// TIA Portal V20 export
DATA_BLOCK "DB_Tracability"   // DB94
// stored: InstanceOfName FB_Tracability, InstanceOfType FB
"FB_Tracability"
   // VAR_INPUT
   //    iCondTransfertExtInTo1 : Bool;
   //    iCondTransfertExtInTo2 : Bool;
   //    iCondTransfert1To3 : Bool;
   //    iCondTransfert2To3 : Bool;
   //    iCondTransfert3To4 : Bool;
   //    iCondTransfert4To5 : Bool;
   //    iCondTransfert5To6 : Bool;
   //    iCondTransfert5To7 : Bool;
   //    iCondTransfert6ToExtOut : Bool;
   //    iCondTransfert7ToExtOut : Bool;
   // END_VAR
   // VAR
   //    sRT_ConditionExtInTo1 : R_TRIG;
   //    sRT_ConditionExtInTo2 { S7_SetPoint := 'True'} : R_TRIG;
   //    sRT_Condition1To3 { S7_SetPoint := 'True'} : R_TRIG;
   //    sRT_Condition2To3 { S7_SetPoint := 'True'} : R_TRIG;
   //    sRT_Condition3To4 { S7_SetPoint := 'True'} : R_TRIG;
   //    sRT_Condition4To5 { S7_SetPoint := 'True'} : R_TRIG;
   //    sRT_Condition5To6 { S7_SetPoint := 'True'} : R_TRIG;
   //    sRT_Condition5To7 { S7_SetPoint := 'True'} : R_TRIG;
   //    sRT_Condition6ToExtOut { S7_SetPoint := 'True'} : R_TRIG;
   //    sRT_Condition7ToExtOut { S7_SetPoint := 'True'} : R_TRIG;
   //    sIndex : Int;
   //    sCheckTransfertExtInTo1 : Bool;
   //    sCheckTransfertExtInTo2 : Bool;
   //    sCheckTransfert1To3 : Bool;
   //    sCheckTransfert2To3 : Bool;
   //    sCheckTransfert3To4 : Bool;
   //    sCheckTransfert4To5 : Bool;
   //    sCheckTransfert5To6 : Bool;
   //    sCheckTransfert5To7 : Bool;
   //    sCheckTransfert6ToExtOut : Bool;
   //    sCheckTransfert7ToExtOut : Bool;
   //    sLaserTime : "FB_TimeCounter";
   //    sMemoPartDMC { S7_SetPoint := 'True'} : Array[0..19] of Byte;
   // END_VAR
   // VAR RETAIN
   //    sIEC_CounterCycleLaser { S7_SetPoint := 'True'} : TONR_TIME;
   //    sIEC_CounterCycleTime { S7_SetPoint := 'True'} : TONR_TIME;
   //    sStartCounterCycleLaser { S7_SetPoint := 'True'} : Bool;
   //    sStartCounterCycleTime { S7_SetPoint := 'True'} : Bool;
   // END_VAR
BEGIN
END_DATA_BLOCK
